// TIA Portal project "Wshing machine 2 timers" (V16)

(* hardware
DEVICE "S7-1200 station_1"  S7-1200 Station
   slot 0: "Rack_0"  S7-1200 Rack  Rack  V1.0
   slot 1: "PLC_1"  CPU 1212C AC/DC/Rly  6ES7 212-1BE40-0XB0  V4.0
*)

// ===== PLC "PLC_1"  CPU 1212C AC/DC/Rly =====

VAR_GLOBAL   // PLC tag table "Default tag table"
   "start" AT %I0.2 : Bool;
   "stop" AT %I0.3 : Bool;
   "kmF" AT %Q0.0 : Bool;
   "kmR" AT %Q0.1 : Bool;
   "km3" AT %Q0.2 : Bool;
   "km4" AT %Q0.3 : Bool;
   "loop marker" AT %M0.0 : Bool;
   "Tag_1" AT %M0.1 : Bool;
END_VAR

// folder: System blocks/Program resources

DATA_BLOCK "T1"   // DB1
{ S7_Optimized_Access := 'TRUE' }
AUTHOR : Simatic
FAMILY : IEC
NAME : IEC_TMR
VERSION : 1.0
// stored: InstanceOfName IEC_TIMER
"IEC_TIMER"
BEGIN
END_DATA_BLOCK

DATA_BLOCK "T2"   // DB2
{ S7_Optimized_Access := 'TRUE' }
AUTHOR : Simatic
FAMILY : IEC
NAME : IEC_TMR
VERSION : 1.0
// stored: InstanceOfName IEC_TIMER
"IEC_TIMER"
BEGIN
END_DATA_BLOCK

DATA_BLOCK "C1"   // DB3
{ S7_Optimized_Access := 'TRUE' }
AUTHOR : Simatic
FAMILY : IEC
NAME : CNTR
VERSION : 1.0
// stored: InstanceOfName IEC_COUNTER
"IEC_COUNTER"
BEGIN
END_DATA_BLOCK

// folder: (top level)

ORGANIZATION_BLOCK "Main"   // OB1, LAD, ProgramCycle
TITLE = "Main Program Sweep (Cycle)"
{ S7_Optimized_Access := 'TRUE' }
VERSION : 0.1
   VAR_INPUT
      Initial_Call : Bool;   // Initial call of this OB
      Remanence : Bool;   // =True, if remanent data are available
   END_VAR
BEGIN

REGION Network 1
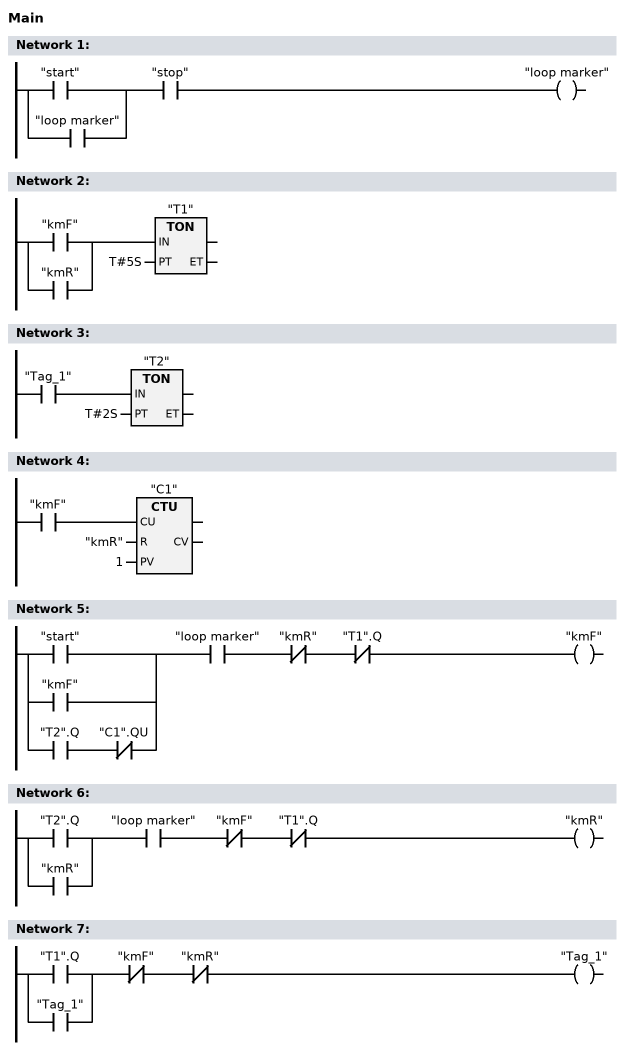
   RUNG wire#powerrail
      Contact( "start" )
      wire#w1
      Contact( "stop" )
      Coil( "loop marker" )
   END_RUNG
   RUNG wire#powerrail
      Contact( "loop marker" )
   END_RUNG wire#w1
   // the same network as SCL:
   "loop marker" := ("start" OR "loop marker") AND "stop";
END_REGION

REGION Network 2
   "T1".TON(IN := "kmF" OR "kmR", PT := T#5S);
END_REGION

REGION Network 3
   "T2".TON(IN := "Tag_1", PT := T#2S);
END_REGION

REGION Network 4
   "C1".CTU(CU := "kmF", R := "kmR", PV := 1);
END_REGION

REGION Network 5
   RUNG wire#powerrail
      Contact( "start" )
      wire#w1
      Contact( "loop marker" )
      I_Contact( "kmR" )
      I_Contact( "T1".Q )
      Coil( "kmF" )
   END_RUNG
   RUNG wire#powerrail
      Contact( "kmF" )
   END_RUNG wire#w1
   RUNG wire#powerrail
      Contact( "T2".Q )
      I_Contact( "C1".QU )
   END_RUNG wire#w1
   // the same network as SCL:
   "kmF" := ("start" OR "kmF" OR ("T2".Q AND NOT "C1".QU)) AND "loop marker" AND NOT "kmR" AND NOT "T1".Q;
END_REGION

REGION Network 6
   RUNG wire#powerrail
      Contact( "T2".Q )
      wire#w1
      Contact( "loop marker" )
      I_Contact( "kmF" )
      I_Contact( "T1".Q )
      Coil( "kmR" )
   END_RUNG
   RUNG wire#powerrail
      Contact( "kmR" )
   END_RUNG wire#w1
   // the same network as SCL:
   "kmR" := ("T2".Q OR "kmR") AND "loop marker" AND NOT "kmF" AND NOT "T1".Q;
END_REGION

REGION Network 7
   RUNG wire#powerrail
      Contact( "T1".Q )
      wire#w1
      I_Contact( "kmF" )
      I_Contact( "kmR" )
      Coil( "Tag_1" )
   END_RUNG
   RUNG wire#powerrail
      Contact( "Tag_1" )
   END_RUNG wire#w1
   // the same network as SCL:
   "Tag_1" := ("T1".Q OR "Tag_1") AND NOT "kmF" AND NOT "kmR";
END_REGION
END_ORGANIZATION_BLOCK